// Mitsubishi GX Works2 project: timer2   PLC: Q03UDV

PROGRAM MAIN
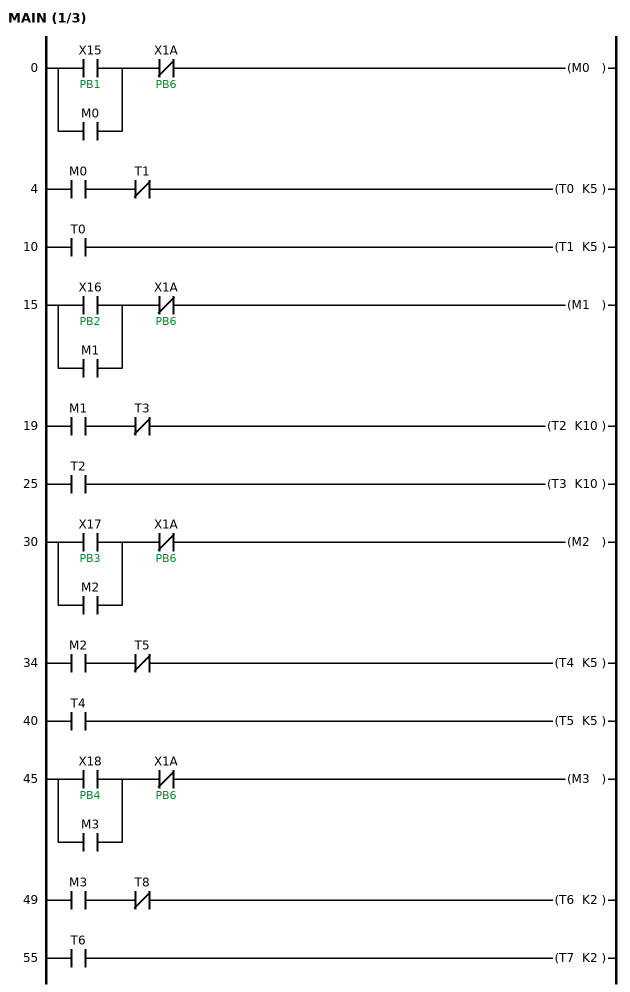
0     LD      X15  ; PB1
      OR      M0
      ANI     X1A  ; PB6
      OUT     M0
4     LD      M0
      ANI     T1
      OUT     T0 K5
10    LD      T0
      OUT     T1 K5
15    LD      X16  ; PB2
      OR      M1
      ANI     X1A  ; PB6
      OUT     M1
19    LD      M1
      ANI     T3
      OUT     T2 K10
25    LD      T2
      OUT     T3 K10
30    LD      X17  ; PB3
      OR      M2
      ANI     X1A  ; PB6
      OUT     M2
34    LD      M2
      ANI     T5
      OUT     T4 K5
40    LD      T4
      OUT     T5 K5
45    LD      X18  ; PB4
      OR      M3
      ANI     X1A  ; PB6
      OUT     M3
49    LD      M3
      ANI     T8
      OUT     T6 K2
55    LD      T6
      OUT     T7 K2
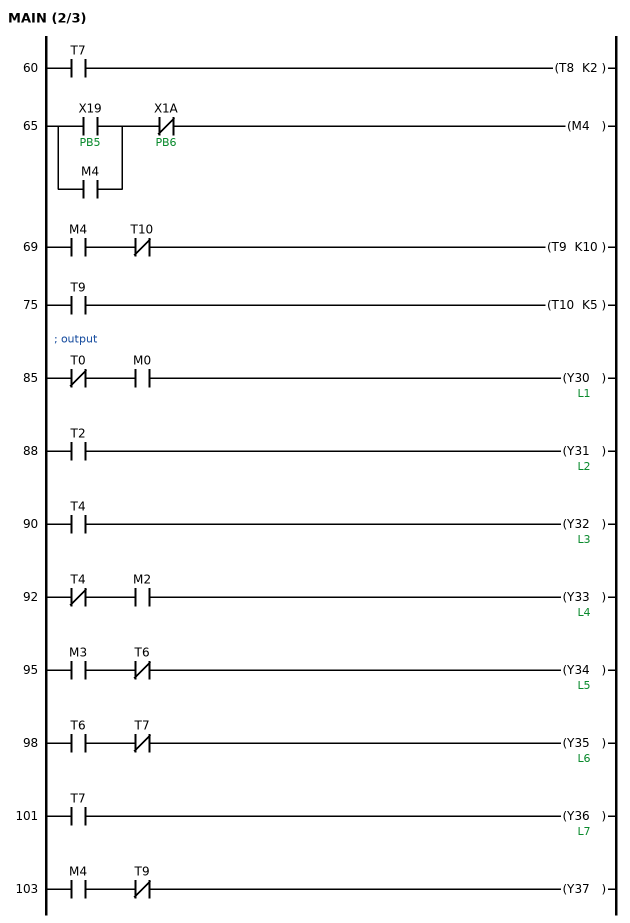
60    LD      T7
      OUT     T8 K2
65    LD      X19  ; PB5
      OR      M4
      ANI     X1A  ; PB6
      OUT     M4
69    LD      M4
      ANI     T10
      OUT     T9 K10
75    LD      T9
      OUT     T10 K5
; output
85    LDI     T0
      AND     M0
      OUT     Y30  ; L1
88    LD      T2
      OUT     Y31  ; L2
90    LD      T4
      OUT     Y32  ; L3
92    LDI     T4
      AND     M2
      OUT     Y33  ; L4
95    LD      M3
      ANI     T6
      OUT     Y34  ; L5
98    LD      T6
      ANI     T7
      OUT     Y35  ; L6
101   LD      T7
      OUT     Y36  ; L7
103   LD      M4
      ANI     T9
      OUT     Y37
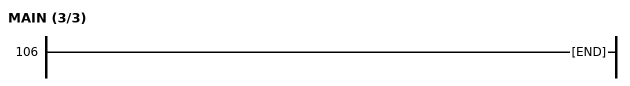
106   END
END_PROGRAM

// device comments not shown above
X1  ; RS1-1
X2  ; RS1-2
X3  ; RS2-1
X4  ; RS2-2
X1B  ; PB7
X1C  ; PB8
Y38  ; SV1-1
Y39  ; SV1-2
Y3A  ; SV2
Y3B  ; SV3
